{attribute 'hide_all_locals'}
FUNCTION_BLOCK PositionTrigger EXTENDS Objective

VAR
	internalTrackPosition		: LREAL;
	internalTriggerDirection	: Tc2_MC2.MC_Direction;
	internalMoverPastPosition	: BOOL;
	internalCurrentMover		: POINTER TO Mover;
	someMoverPast				: BOOL;
	whichMover					: INT;
	i							: INT;
	moverLastPos				: ARRAY[0..GVL.NUM_MOVERS-1] OF LREAL;		// Positions of tracked movers from last cycle
	moverLastTurns				: ARRAY[0..GVL.NUM_MOVERS-1] OF DINT;		// Turn count of tracked movers from last cycle
	positiveRolloverDetected	: BOOL;
	negativeRolloverDetected	: BOOL;
END_VAR

{attribute 'monitoring' := 'variable'}
PROPERTY CurrentMover : REFERENCE TO Mover
GET


CurrentMover	REF= internalCurrentMover^;
	
// If the Trigger has no CurrentMover, then return an imposter ErrorMover, whose method calls all trigger an error message
IF __ISVALIDREF( CurrentMover ) = FALSE THEN	
	ErrorMover.SourceInstancePath	:= THIS^.InstancePath;
	CurrentMover	REF= ErrorMover;
END_IF
END_GET
END_PROPERTY

METHOD Cyclic : BOOL
VAR_INPUT
END_VAR


someMoverPast		:= FALSE;
whichMover			:= 0;


FOR i := 0 TO GVL.NUM_MOVERS-1 DO	
	IF internalTrackedMovers[i] <> 0 THEN
		
	
		
	
	
		// Determine if a position rollover occured in the last cycle
		IF internalTrackedMovers[i]^.AxisReference.NcToPlc.ModuloActTurns > moverLastTurns[i] THEN
			positiveRolloverDetected		:= TRUE;
		ELSIF internalTrackedMovers[i]^.AxisReference.NcToPlc.ModuloActTurns < moverLastTurns[i] THEN
			negativeRolloverDetected		:= TRUE;
		ELSE
			positiveRolloverDetected		:= FALSE;
			negativeRolloverDetected		:= FALSE;
		END_IF
		// Set value for next cycle
		moverLastTurns[i]	:= internalTrackedMovers[i]^.AxisReference.NcToPlc.ModuloActTurns;
	
		
		// Can combine with above stanza
		IF positiveRolloverDetected THEN
			moverLastPos[i]		:= moverLastPos[i] - GVL.TRACK_LENGTH;
		ELSIF negativeRolloverDetected THEN
			moverLastPos[i]		:= moverLastPos[i] + GVL.TRACK_LENGTH;				
		END_IF
		
		
		
		
		
		
		// Watch for movers crossing the threshold position
		IF TriggerDirection = MC_Positive_Direction THEN
			
			IF moverLastPos[i] < internalTrackPosition AND
				internalTrackedMovers[i]^.AxisReference.NcToPlc.ModuloActPos >= internalTrackPosition THEN
				// Position trigger event detected
				someMoverPast	:= TRUE;
				whichMover		:= i;
			END_IF
			
		ELSIF TriggerDirection = MC_Negative_Direction THEN
			
			IF moverLastPos[i] > internalTrackPosition AND
				internalTrackedMovers[i]^.AxisReference.NcToPlc.ModuloActPos <= internalTrackPosition THEN
				// Position trigger event detected
				someMoverPast	:= TRUE;
				whichMover		:= i;
			END_IF		
		
		END_IF

		
		
		moverLastPos[i]			:= internalTrackedMovers[i]^.AxisReference.NcToPlc.ModuloActPos;
		
		
		
		
	ELSE
		IF TriggerDirection = MC_Negative_Direction THEN
			moverLastPos[i]		:= -1E300;	// very negative value, to prevent false-positive triggers on first cycle
		ELSIF TriggerDirection = MC_Positive_Direction THEN
			moverLastPos[i]		:= 1E300;	// very positive value, to prevent false-positive triggers on first cycle
		END_IF
	END_IF

	
	
	
	
END_FOR




IF someMoverPast THEN
	internalMoverPastPosition		:= TRUE;
	internalCurrentMover			:= internalTrackedMovers[whichMover];
ELSE
	internalMoverPastPosition		:= FALSE;
	internalCurrentMover			:= 0;		
END_IF
END_METHOD

{attribute 'monitoring' := 'variable'}
PROPERTY MoverPassedPosition : BOOL
GET

	MoverPassedPosition	:= internalMoverPastPosition;
END_GET
END_PROPERTY

{attribute 'monitoring' := 'call'}
PROPERTY TrackPosition : LREAL
GET


	TrackPosition	:= internalTrackPosition;
END_GET
SET


	// todo maybe do a limits check here?
	internalTrackPosition	:= TrackPosition;
END_SET
END_PROPERTY

{attribute 'monitoring' := 'call'}
PROPERTY TriggerDirection : Tc2_MC2.MC_Direction
GET
END_GET
SET
END_SET
END_PROPERTY

END_FUNCTION_BLOCK

(* stored: Version 1.1.0.1, ProductVersion 3.1.4024.9
   POU PositionTrigger: Id {2be242dd-21c3-49cc-ab16-707ac1bbd2e6}, SpecialFunc None
   Folder Methods: Id {5543ded2-7a48-48d8-8a29-b553779a4150}
   Folder Properties: Id {8d51ba54-c5eb-42a0-ba8e-ec7acb9ee6ae}
   Property CurrentMover: Id {08e03357-929c-40a3-8446-c462dfedb470}
   Get Get: Id {d772a5d5-0e79-4d5f-ad7a-159060b39ae3}
   Method Cyclic: Id {837bb22f-75d9-4f81-992f-274e662e1a69}
   Property MoverPassedPosition: Id {6ef1f07f-a5fa-461a-8898-d87506fab1a7}
   Get Get: Id {a91db2b1-564e-4fdf-92fa-febfe2148c87}
   Property TrackPosition: Id {ec302377-0190-40b3-b726-4713ec7a403b}
   Get Get: Id {ff32a52e-c366-4283-94bb-898d1069bf0a}
   Set Set: Id {b77ff2fd-1ee8-41cd-8d5f-9b4c152df435}
   Property TriggerDirection: Id {da3896fd-b18b-47dc-bafd-92a621ffa675}
   Get Get: Id {423fc284-e969-4051-9911-5a30b9185b1a}
   Set Set: Id {f583cf2c-e716-4e32-994c-ff6c210917d6} *)
